# EPICS autosave request: delaygen/delaygenApp/Db/drvDG645_settings.req
$(P)$(R)Label

$(P)$(R)ADelayTweakAO
$(P)$(R)BDelayTweakAO
$(P)$(R)CDelayTweakAO
$(P)$(R)DDelayTweakAO
$(P)$(R)EDelayTweakAO
$(P)$(R)FDelayTweakAO
$(P)$(R)GDelayTweakAO
$(P)$(R)HDelayTweakAO

$(P)$(R)T0OutputAmpTweakAO
$(P)$(R)ABOutputAmpTweakAO
$(P)$(R)CDOutputAmpTweakAO
$(P)$(R)EFOutputAmpTweakAO
$(P)$(R)GHOutputAmpTweakAO

$(P)$(R)T0OutputOffsetTweakAO
$(P)$(R)ABOutputOffsetTweakAO
$(P)$(R)CDOutputOffsetTweakAO
$(P)$(R)EFOutputOffsetTweakAO
$(P)$(R)GHOutputOffsetTweakAO

$(P)$(R)IfaceIpAddrSO
$(P)$(R)IfaceNetMaskSO
$(P)$(R)IfaceGatewaySO
